FUNCTION_BLOCK NEW_FB_0
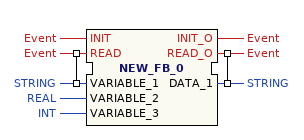
  EVENT_INPUT
    INIT;
    READ WITH VARIABLE_1, , ;
  END_EVENT
  EVENT_OUTPUT
    INIT_O;
    READ_O WITH DATA_1;
  END_EVENT
  VAR_INPUT
    VARIABLE_1 : STRING;
    VARIABLE_2 : REAL;
    VARIABLE_3 : INT;
  END_VAR
  VAR_OUTPUT
    DATA_1 : STRING;
  END_VAR
END_FUNCTION_BLOCK
